ABB RobotStudio station: Welding_2.rspag

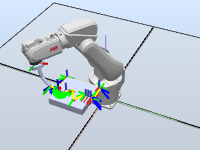
--- station ---
Station Welding_1 (saved by RobotStudio 20.1.9014.1)
Controller Controller2
  mechanical unit ROB_1: IRB120_3_58__01, 6 joints, base frame (0, 0, 0) mm
Layout (positions relative to the parent item):
  - IRB120_3_58__01 [mechanism, from Robots\IRB120_3_58_G_01.rslib] at (0, 0, 0) mm; joint values [-0.5429, 0.6455, -0.6027, 0.2244, 1.6631, 1.0335] (rad or m)
  - AssemblyWeldingTorch (2)_2 [part] at (431.78, -161.71, 537.76) mm, rotated rx -105 ry 0 rz -180 deg
  - Task1_Part1_2 [part] at (400, -100, 350) mm, rotated rx 90 ry 0 rz 0 deg
  - Task1_Part2 [part] at (300, -100, 350) mm, rotated rx 90 ry 0 rz 0 deg
  - Frame_1 [frame] at (400, 100, 370) mm
  - Frame_5 [frame] at (300, 100, 370) mm
  - Frame_6 [frame] at (300, -100, 370) mm
  - Frame_9 [frame] at (400, 85, 370) mm
  - Frame_10 [frame] at (400, 70, 370) mm
  - Frame_11 [frame] at (400, -50, 370) mm
Attachment: AssemblyWeldingTorch (2)_2 is attached to IRB120_3_58__01 / Link6

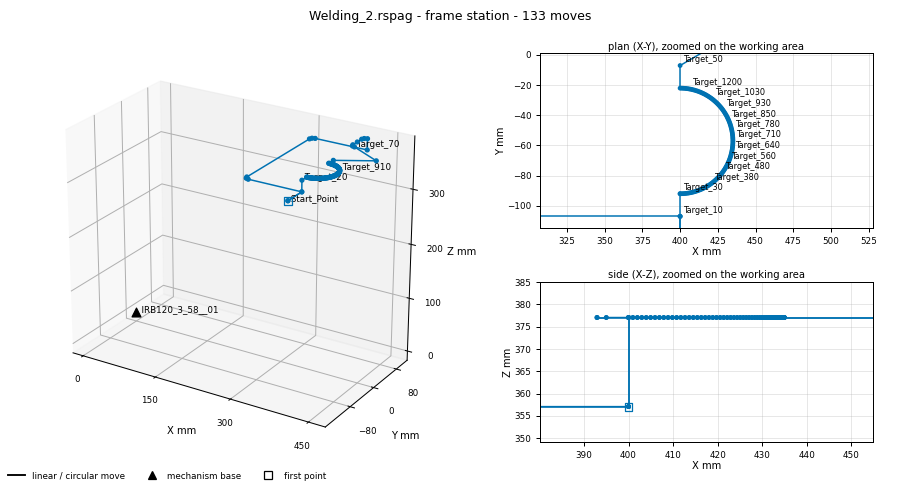
[picture p0: tool path of Welding_2.rspag in frame station, 133 of 133 moves have a stored position in this frame; points joined in program order, loops and branches not executed]
--- Backups/Controller2/RAPID/TASK1/PROGMOD/CalibData.mod ---
MODULE CalibData
    TASK PERS tooldata Tooldata_1:=[TRUE,[[35,0,150.231],[0.866025404,0,-0.5,0]],[1,[0,0,1],[1,0,0,0],0,0,0]];
    TASK PERS wobjdata weldPlate_1:=[FALSE,TRUE,"",[[400,-100,350],[1,0,0,0]],[[0,0,0],[1,0,0,0]]];
ENDMODULE

--- Backups/Controller2/RAPID/TASK1/PROGMOD/Module1.mod ---
MODULE Module1
        CONST robtarget Start_Point:=[[0,-50,7.071067812],[0.27059805,0.653281482,0.653281482,-0.27059805],[-1,0,0,0],[9E+09,9E+09,9E+09,9E+09,9E+09,9E+09]];
    CONST robtarget Target_10:=[[0,-7.071,7.071067812],[0.27059805,0.653281482,0.653281482,-0.27059805],[-1,0,0,0],[9E+09,9E+09,9E+09,9E+09,9E+09,9E+09]];
    CONST robtarget Target_20:=[[0,-7.071,27.071067812],[0.27059805,0.653281482,0.653281482,-0.27059805],[-1,0,0,0],[9E+09,9E+09,9E+09,9E+09,9E+09,9E+09]];
    CONST robtarget Target_30:=[[0,7.929,27.071067812],[0.27059805,0.653281482,0.653281482,-0.27059805],[-1,0,0,0],[9E+09,9E+09,9E+09,9E+09,9E+09,9E+09]];
    CONST robtarget Target_40:=[[0,77.929,27.071067812],[0.27059805,0.653281482,0.653281482,-0.27059805],[-1,0,0,0],[9E+09,9E+09,9E+09,9E+09,9E+09,9E+09]];
    CONST robtarget Target_50:=[[0,92.929,27.071067812],[0.27059805,0.653281482,0.653281482,-0.27059805],[-1,0,0,0],[9E+09,9E+09,9E+09,9E+09,9E+09,9E+09]];
    CONST robtarget Target_60:=[[60,127.929,27.071067812],[0.27059805,0.653281482,0.653281482,-0.27059805],[-1,0,0,0],[9E+09,9E+09,9E+09,9E+09,9E+09,9E+09]];
    CONST robtarget Target_70:=[[0,162.929,27.071067812],[0.27059805,0.653281482,0.653281482,-0.27059805],[-1,0,0,0],[9E+09,9E+09,9E+09,9E+09,9E+09,9E+09]];
    CONST robtarget Target_90:=[[0,207.071,7.071067812],[0.27059805,-0.653281482,0.653281482,0.27059805],[0,-1,3,0],[9E+09,9E+09,9E+09,9E+09,9E+09,9E+09]];
    CONST robtarget Target_100:=[[-100,207.071,7.071067812],[0.27059805,-0.653281482,0.653281482,0.27059805],[0,-1,3,0],[9E+09,9E+09,9E+09,9E+09,9E+09,9E+09]];
    CONST robtarget Target_110:=[[-107.071,200,7.071067812],[0,0.923879532,0,-0.382683432],[0,-1,2,0],[9E+09,9E+09,9E+09,9E+09,9E+09,9E+09]];
    CONST robtarget Target_120:=[[-107.071,0,7.071],[0,0.923879533,0,-0.382683432],[-1,0,1,0],[9E+09,9E+09,9E+09,9E+09,9E+09,9E+09]];
    CONST robtarget Target_130:=[[-100,-7.071,7.071],[0.27059805,0.653281483,0.653281483,-0.27059805],[-1,0,0,0],[9E+09,9E+09,9E+09,9E+09,9E+09,9E+09]];
    CONST robtarget Target_140:=[[0,-7.071,7.071067812],[0.27059805,0.653281482,0.653281482,-0.27059805],[-1,0,0,0],[9E+09,9E+09,9E+09,9E+09,9E+09,9E+09]];
    CONST robtarget Target_150:=[[-2,-9.698,8.29],[0.699810239,0.292325175,0.577022876,0.303077913],[-1,0,-1,0],[9E+09,9E+09,9E+09,9E+09,9E+09,9E+09]];
    CONST robtarget End_Point:=[[0,-50,0],[0.27059805,0.653281482,0.653281482,-0.27059805],[-1,0,0,0],[9E+09,9E+09,9E+09,9E+09,9E+09,9E+09]];
    CONST robtarget Target_30_1:=[[35,42.928932188,27.071067812],[0.27059805,0.653281482,0.653281482,-0.27059805],[-1,0,0,0],[9E+09,9E+09,9E+09,9E+09,9E+09,9E+09]];
    CONST robtarget Target_30_4:=[[32.122,36.212,30],[0.699810239,0.292325175,0.577022876,0.303077913],[-1,0,-1,0],[9E+09,9E+09,9E+09,9E+09,9E+09,9E+09]];
    CONST robtarget Target_30_5:=[[26.122,57.788,30],[0.699810239,0.292325175,0.577022876,0.303077913],[-1,0,-1,0],[9E+09,9E+09,9E+09,9E+09,9E+09,9E+09]];
    CONST robtarget Target_30_6:=[[7.364,71.822,30],[0.699810239,0.292325175,0.577022876,0.303077913],[-1,0,-1,0],[9E+09,9E+09,9E+09,9E+09,9E+09,9E+09]];
    CONST robtarget Target_30_7:=[[-2.5,81.534,30],[0.699810239,0.292325175,0.577022876,0.303077913],[-1,0,-1,0],[9E+09,9E+09,9E+09,9E+09,9E+09,9E+09]];
    CONST robtarget Target_30_8:=[[-2.5,88,30],[0.699810239,0.292325175,0.577022876,0.303077913],[-1,0,-1,0],[9E+09,9E+09,9E+09,9E+09,9E+09,9E+09]];
    CONST robtarget Target_30_3:=[[27.364,20.178,30],[0.699810239,0.292325175,0.577022876,0.303077913],[-1,0,-1,0],[9E+09,9E+09,9E+09,9E+09,9E+09,9E+09]];
    CONST robtarget Target_80:=[[-7.071067812,200,27.071],[0,0.923879532,0,-0.382683432],[0,-1,2,0],[9E+09,9E+09,9E+09,9E+09,9E+09,9E+09]];
    CONST robtarget Target_30_2:=[[15.186,8.466,30],[0.699810239,0.292325175,0.577022876,0.303077913],[-1,0,-1,0],[9E+09,9E+09,9E+09,9E+09,9E+09,9E+09]];
    CONST robtarget Target_70_2:=[[-5,165.000095901,27.071],[0.146446609,0.853553391,0.353553391,-0.35355339],[0,0,1,0],[9E+09,9E+09,9E+09,9E+09,9E+09,9E+09]];
    CONST robtarget Target_70_2_2:=[[-7.071,170.000067812,27.071],[0,0.923879533,0,-0.382683432],[0,-1,2,0],[9E+09,9E+09,9E+09,9E+09,9E+09,9E+09]];
    CONST robtarget Target_70_3:=[[-7.071067812,185,27.071],[0,0.923879533,0,-0.382683432],[0,-1,2,0],[9E+09,9E+09,9E+09,9E+09,9E+09,9E+09]];
    CONST robtarget Target_80_3:=[[-5,205,27.071],[0.146446609,-0.853553391,0.353553391,0.353553391],[0,-1,2,0],[9E+09,9E+09,9E+09,9E+09,9E+09,9E+09]];
    CONST robtarget Target_80_4:=[[0,207.071067812,27.071],[0.27059805,-0.653281482,0.653281482,0.27059805],[0,-1,3,0],[9E+09,9E+09,9E+09,9E+09,9E+09,9E+09]];
    CONST robtarget Target_100_3:=[[-104.99995205,204.99995205,7.071067812],[0.146446609,-0.853553391,0.353553391,0.353553391],[0,-1,2,0],[9E+09,9E+09,9E+09,9E+09,9E+09,9E+09]];
    CONST robtarget Target_120_3:=[[-104.99995205,-4.99995205,7.071],[0.146446609,0.853553391,0.353553391,-0.35355339],[-1,0,1,0],[9E+09,9E+09,9E+09,9E+09,9E+09,9E+09]];
    CONST robtarget zEnd_Point:=[[0,-50,7.071067812],[0.27059805,0.653281482,0.653281482,-0.27059805],[-1,0,0,0],[9E+09,9E+09,9E+09,9E+09,9E+09,9E+09]];
    CONST robtarget Target_170:=[[0.999863951,7.94321693,27.071067812],[0.27059805,0.653281482,0.653281482,-0.27059805],[-1,0,0,0],[9E+09,9E+09,9E+09,9E+09,9E+09,9E+09]];
    CONST robtarget Target_180:=[[1.998911742,7.986059498,27.071067812],[0.27059805,0.653281482,0.653281482,-0.27059805],[-1,0,0,0],[9E+09,9E+09,9E+09,9E+09,9E+09,9E+09]];
    CONST robtarget Target_190:=[[2.99632788,8.057424919,27.071067812],[0.27059805,0.653281482,0.653281482,-0.27059805],[-1,0,0,0],[9E+09,9E+09,9E+09,9E+09,9E+09,9E+09]];
    CONST robtarget Target_200:=[[3.991298202,8.15725494,27.071067812],[0.27059805,0.653281482,0.653281482,-0.27059805],[-1,0,0,0],[9E+09,9E+09,9E+09,9E+09,9E+09,9E+09]];
    CONST robtarget Target_210:=[[4.983010543,8.285468072,27.071067812],[0.27059805,0.653281482,0.653281482,-0.27059805],[-1,0,0,0],[9E+09,9E+09,9E+09,9E+09,9E+09,9E+09]];
    CONST robtarget Target_220:=[[5.970655397,8.44195966,27.071067812],[0.27059805,0.653281482,0.653281482,-0.27059805],[-1,0,0,0],[9E+09,9E+09,9E+09,9E+09,9E+09,9E+09]];
    CONST robtarget Target_230:=[[6.953426578,8.626601964,27.071067812],[0.27059805,0.653281482,0.653281482,-0.27059805],[-1,0,0,0],[9E+09,9E+09,9E+09,9E+09,9E+09,9E+09]];
    CONST robtarget Target_240:=[[7.930521878,8.839244264,27.071067812],[0.27059805,0.653281482,0.653281482,-0.27059805],[-1,0,0,0],[9E+09,9E+09,9E+09,9E+09,9E+09,9E+09]];
    CONST robtarget Target_250:=[[8.901143724,9.079712989,27.071067812],[0.27059805,0.653281482,0.653281482,-0.27059805],[-1,0,0,0],[9E+09,9E+09,9E+09,9E+09,9E+09,9E+09]];
    CONST robtarget Target_260:=[[9.864499824,9.347811849,27.071067812],[0.27059805,0.653281482,0.653281482,-0.27059805],[-1,0,0,0],[9E+09,9E+09,9E+09,9E+09,9E+09,9E+09]];
    CONST robtarget Target_270:=[[10.819803819,9.643322004,27.071067812],[0.27059805,0.653281482,0.653281482,-0.27059805],[-1,0,0,0],[9E+09,9E+09,9E+09,9E+09,9E+09,9E+09]];
    CONST robtarget Target_280:=[[11.766275922,9.966002237,27.071067812],[0.27059805,0.653281482,0.653281482,-0.27059805],[-1,0,0,0],[9E+09,9E+09,9E+09,9E+09,9E+09,9E+09]];
    CONST robtarget Target_290:=[[12.703143555,10.315589155,27.071067812],[0.27059805,0.653281482,0.653281482,-0.27059805],[-1,0,0,0],[9E+09,9E+09,9E+09,9E+09,9E+09,9E+09]];
    CONST robtarget Target_300:=[[13.629641981,10.691797398,27.071067812],[0.27059805,0.653281482,0.653281482,-0.27059805],[-1,0,0,0],[9E+09,9E+09,9E+09,9E+09,9E+09,9E+09]];
    CONST robtarget Target_310:=[[14.545014925,11.094319879,27.071067812],[0.27059805,0.653281482,0.653281482,-0.27059805],[-1,0,0,0],[9E+09,9E+09,9E+09,9E+09,9E+09,9E+09]];
    CONST robtarget Target_320:=[[15.448515195,11.522828032,27.071067812],[0.27059805,0.653281482,0.653281482,-0.27059805],[-1,0,0,0],[9E+09,9E+09,9E+09,9E+09,9E+09,9E+09]];
    CONST robtarget Target_330:=[[16.33940529,11.976972076,27.071067812],[0.27059805,0.653281482,0.653281482,-0.27059805],[-1,0,0,0],[9E+09,9E+09,9E+09,9E+09,9E+09,9E+09]];
    CONST robtarget Target_340:=[[17.216958002,12.456381308,27.071067812],[0.27059805,0.653281482,0.653281482,-0.27059805],[-1,0,0,0],[9E+09,9E+09,9E+09,9E+09,9E+09,9E+09]];
    CONST robtarget Target_350:=[[18.080457011,12.960664399,27.071067812],[0.27059805,0.653281482,0.653281482,-0.27059805],[-1,0,0,0],[9E+09,9E+09,9E+09,9E+09,9E+09,9E+09]];
    CONST robtarget Target_360:=[[18.929197468,13.489409718,27.071067812],[0.27059805,0.653281482,0.653281482,-0.27059805],[-1,0,0,0],[9E+09,9E+09,9E+09,9E+09,9E+09,9E+09]];
    CONST robtarget Target_370:=[[19.762486569,14.042185666,27.071067812],[0.27059805,0.653281482,0.653281482,-0.27059805],[-1,0,0,0],[9E+09,9E+09,9E+09,9E+09,9E+09,9E+09]];
    CONST robtarget Target_380:=[[20.579644125,14.618541027,27.071067812],[0.27059805,0.653281482,0.653281482,-0.27059805],[-1,0,0,0],[9E+09,9E+09,9E+09,9E+09,9E+09,9E+09]];
    CONST robtarget Target_390:=[[21.380003115,15.21800534,27.071067812],[0.27059805,0.653281482,0.653281482,-0.27059805],[-1,0,0,0],[9E+09,9E+09,9E+09,9E+09,9E+09,9E+09]];
    CONST robtarget Target_400:=[[22.162910229,15.840089278,27.071067812],[0.27059805,0.653281482,0.653281482,-0.27059805],[-1,0,0,0],[9E+09,9E+09,9E+09,9E+09,9E+09,9E+09]];
    CONST robtarget Target_410:=[[22.927726401,16.484285053,27.071067812],[0.27059805,0.653281482,0.653281482,-0.27059805],[-1,0,0,0],[9E+09,9E+09,9E+09,9E+09,9E+09,9E+09]];
    CONST robtarget Target_420:=[[23.673827336,17.150066827,27.071067812],[0.27059805,0.653281482,0.653281482,-0.27059805],[-1,0,0,0],[9E+09,9E+09,9E+09,9E+09,9E+09,9E+09]];
    CONST robtarget Target_430:=[[24.400604011,17.836891141,27.071067812],[0.27059805,0.653281482,0.653281482,-0.27059805],[-1,0,0,0],[9E+09,9E+09,9E+09,9E+09,9E+09,9E+09]];
    CONST robtarget Target_440:=[[25.107463181,18.544197361,27.071067812],[0.27059805,0.653281482,0.653281482,-0.27059805],[-1,0,0,0],[9E+09,9E+09,9E+09,9E+09,9E+09,9E+09]];
    CONST robtarget Target_450:=[[25.793827858,19.271408132,27.071067812],[0.27059805,0.653281482,0.653281482,-0.27059805],[-1,0,0,0],[9E+09,9E+09,9E+09,9E+09,9E+09,9E+09]];
    CONST robtarget Target_460:=[[26.45913778,20.017929854,27.071067812],[0.27059805,0.653281482,0.653281482,-0.27059805],[-1,0,0,0],[9E+09,9E+09,9E+09,9E+09,9E+09,9E+09]];
    CONST robtarget Target_470:=[[27.102849876,20.783153163,27.071067812],[0.27059805,0.653281482,0.653281482,-0.27059805],[-1,0,0,0],[9E+09,9E+09,9E+09,9E+09,9E+09,9E+09]];
    CONST robtarget Target_480:=[[27.724438701,21.566453429,27.071067812],[0.27059805,0.653281482,0.653281482,-0.27059805],[-1,0,0,0],[9E+09,9E+09,9E+09,9E+09,9E+09,9E+09]];
    CONST robtarget Target_490:=[[28.323396871,22.367191267,27.071067812],[0.27059805,0.653281482,0.653281482,-0.27059805],[-1,0,0,0],[9E+09,9E+09,9E+09,9E+09,9E+09,9E+09]];
    CONST robtarget Target_500:=[[28.899235474,23.184713058,27.071067812],[0.27059805,0.653281482,0.653281482,-0.27059805],[-1,0,0,0],[9E+09,9E+09,9E+09,9E+09,9E+09,9E+09]];
    CONST robtarget Target_510:=[[29.451484468,24.018351483,27.071067812],[0.27059805,0.653281482,0.653281482,-0.27059805],[-1,0,0,0],[9E+09,9E+09,9E+09,9E+09,9E+09,9E+09]];
    CONST robtarget Target_520:=[[29.97969307,24.867426066,27.071067812],[0.27059805,0.653281482,0.653281482,-0.27059805],[-1,0,0,0],[9E+09,9E+09,9E+09,9E+09,9E+09,9E+09]];
    CONST robtarget Target_530:=[[30.483430118,25.731243732,27.071067812],[0.27059805,0.653281482,0.653281482,-0.27059805],[-1,0,0,0],[9E+09,9E+09,9E+09,9E+09,9E+09,9E+09]];
    CONST robtarget Target_540:=[[30.962284426,26.609099373,27.071067812],[0.27059805,0.653281482,0.653281482,-0.27059805],[-1,0,0,0],[9E+09,9E+09,9E+09,9E+09,9E+09,9E+09]];
    CONST robtarget Target_550:=[[31.415865119,27.50027642,27.071067812],[0.27059805,0.653281482,0.653281482,-0.27059805],[-1,0,0,0],[9E+09,9E+09,9E+09,9E+09,9E+09,9E+09]];
    CONST robtarget Target_560:=[[31.843801953,28.404047432,27.071067812],[0.27059805,0.653281482,0.653281482,-0.27059805],[-1,0,0,0],[9E+09,9E+09,9E+09,9E+09,9E+09,9E+09]];
    CONST robtarget Target_570:=[[32.245745614,29.319674685,27.071067812],[0.27059805,0.653281482,0.653281482,-0.27059805],[-1,0,0,0],[9E+09,9E+09,9E+09,9E+09,9E+09,9E+09]];
    CONST robtarget Target_580:=[[32.621368009,30.246410781,27.071067812],[0.27059805,0.653281482,0.653281482,-0.27059805],[-1,0,0,0],[9E+09,9E+09,9E+09,9E+09,9E+09,9E+09]];
    CONST robtarget Target_590:=[[32.970362527,31.183499252,27.071067812],[0.27059805,0.653281482,0.653281482,-0.27059805],[-1,0,0,0],[9E+09,9E+09,9E+09,9E+09,9E+09,9E+09]];
    CONST robtarget Target_600:=[[33.292444294,32.130175178,27.071067812],[0.27059805,0.653281482,0.653281482,-0.27059805],[-1,0,0,0],[9E+09,9E+09,9E+09,9E+09,9E+09,9E+09]];
    CONST robtarget Target_610:=[[33.587350404,33.085665817,27.071067812],[0.27059805,0.653281482,0.653281482,-0.27059805],[-1,0,0,0],[9E+09,9E+09,9E+09,9E+09,9E+09,9E+09]];
    CONST robtarget Target_620:=[[33.854840134,34.049191229,27.071067812],[0.27059805,0.653281482,0.653281482,-0.27059805],[-1,0,0,0],[9E+09,9E+09,9E+09,9E+09,9E+09,9E+09]];
    CONST robtarget Target_630:=[[34.09469514,35.019964915,27.071067812],[0.27059805,0.653281482,0.653281482,-0.27059805],[-1,0,0,0],[9E+09,9E+09,9E+09,9E+09,9E+09,9E+09]];
    CONST robtarget Target_640:=[[34.306719635,35.997194463,27.071067812],[0.27059805,0.653281482,0.653281482,-0.27059805],[-1,0,0,0],[9E+09,9E+09,9E+09,9E+09,9E+09,9E+09]];
    CONST robtarget Target_650:=[[34.49074055,36.980082186,27.071067812],[0.27059805,0.653281482,0.653281482,-0.27059805],[-1,0,0,0],[9E+09,9E+09,9E+09,9E+09,9E+09,9E+09]];
    CONST robtarget Target_660:=[[34.646607673,37.967825784,27.071067812],[0.27059805,0.653281482,0.653281482,-0.27059805],[-1,0,0,0],[9E+09,9E+09,9E+09,9E+09,9E+09,9E+09]];
    CONST robtarget Target_670:=[[34.774193775,38.959618989,27.071067812],[0.27059805,0.653281482,0.653281482,-0.27059805],[-1,0,0,0],[9E+09,9E+09,9E+09,9E+09,9E+09,9E+09]];
    CONST robtarget Target_680:=[[34.873394712,39.954652229,27.071067812],[0.27059805,0.653281482,0.653281482,-0.27059805],[-1,0,0,0],[9E+09,9E+09,9E+09,9E+09,9E+09,9E+09]];
    CONST robtarget Target_690:=[[34.944129507,40.952113287,27.071067812],[0.27059805,0.653281482,0.653281482,-0.27059805],[-1,0,0,0],[9E+09,9E+09,9E+09,9E+09,9E+09,9E+09]];
    CONST robtarget Target_700:=[[34.986340424,41.951187966,27.071067812],[0.27059805,0.653281482,0.653281482,-0.27059805],[-1,0,0,0],[9E+09,9E+09,9E+09,9E+09,9E+09,9E+09]];
    CONST robtarget Target_710:=[[34.999993005,42.951060749,27.071067812],[0.27059805,0.653281482,0.653281482,-0.27059805],[-1,0,0,0],[9E+09,9E+09,9E+09,9E+09,9E+09,9E+09]];
    CONST robtarget Target_720:=[[34.985076106,43.950915469,27.071067812],[0.27059805,0.653281482,0.653281482,-0.27059805],[-1,0,0,0],[9E+09,9E+09,9E+09,9E+09,9E+09,9E+09]];
    CONST robtarget Target_730:=[[34.941601905,44.949935973,27.071067812],[0.27059805,0.653281482,0.653281482,-0.27059805],[-1,0,0,0],[9E+09,9E+09,9E+09,9E+09,9E+09,9E+09]];
    CONST robtarget Target_740:=[[34.869605888,45.947306791,27.071067812],[0.27059805,0.653281482,0.653281482,-0.27059805],[-1,0,0,0],[9E+09,9E+09,9E+09,9E+09,9E+09,9E+09]];
    CONST robtarget Target_750:=[[34.769146822,46.942213797,27.071067812],[0.27059805,0.653281482,0.653281482,-0.27059805],[-1,0,0,0],[9E+09,9E+09,9E+09,9E+09,9E+09,9E+09]];
    CONST robtarget Target_760:=[[34.64030671,47.933844878,27.071067812],[0.27059805,0.653281482,0.653281482,-0.27059805],[-1,0,0,0],[9E+09,9E+09,9E+09,9E+09,9E+09,9E+09]];
    CONST robtarget Target_770:=[[34.48319072,48.921390593,27.071067812],[0.27059805,0.653281482,0.653281482,-0.27059805],[-1,0,0,0],[9E+09,9E+09,9E+09,9E+09,9E+09,9E+09]];
    CONST robtarget Target_780:=[[34.297927102,49.904044839,27.071067812],[0.27059805,0.653281482,0.653281482,-0.27059805],[-1,0,0,0],[9E+09,9E+09,9E+09,9E+09,9E+09,9E+09]];
    CONST robtarget Target_790:=[[34.084667081,50.881005502,27.071067812],[0.27059805,0.653281482,0.653281482,-0.27059805],[-1,0,0,0],[9E+09,9E+09,9E+09,9E+09,9E+09,9E+09]];
    CONST robtarget Target_800:=[[33.843584734,51.851475119,27.071067812],[0.27059805,0.653281482,0.653281482,-0.27059805],[-1,0,0,0],[9E+09,9E+09,9E+09,9E+09,9E+09,9E+09]];
    CONST robtarget Target_810:=[[33.574876851,52.814661522,27.071067812],[0.27059805,0.653281482,0.653281482,-0.27059805],[-1,0,0,0],[9E+09,9E+09,9E+09,9E+09,9E+09,9E+09]];
    CONST robtarget Target_820:=[[33.278762769,53.769778492,27.071067812],[0.27059805,0.653281482,0.653281482,-0.27059805],[-1,0,0,0],[9E+09,9E+09,9E+09,9E+09,9E+09,9E+09]];
    CONST robtarget Target_830:=[[32.955484198,54.716046393,27.071067812],[0.27059805,0.653281482,0.653281482,-0.27059805],[-1,0,0,0],[9E+09,9E+09,9E+09,9E+09,9E+09,9E+09]];
    CONST robtarget Target_840:=[[32.605305021,55.652692814,27.071067812],[0.27059805,0.653281482,0.653281482,-0.27059805],[-1,0,0,0],[9E+09,9E+09,9E+09,9E+09,9E+09,9E+09]];
    CONST robtarget Target_850:=[[32.22851108,56.578953199,27.071067812],[0.27059805,0.653281482,0.653281482,-0.27059805],[-1,0,0,0],[9E+09,9E+09,9E+09,9E+09,9E+09,9E+09]];
    CONST robtarget Target_860:=[[31.825409939,57.494071467,27.071067812],[0.27059805,0.653281482,0.653281482,-0.27059805],[-1,0,0,0],[9E+09,9E+09,9E+09,9E+09,9E+09,9E+09]];
    CONST robtarget Target_870:=[[31.396330639,58.397300635,27.071067812],[0.27059805,0.653281482,0.653281482,-0.27059805],[-1,0,0,0],[9E+09,9E+09,9E+09,9E+09,9E+09,9E+09]];
    CONST robtarget Target_880:=[[30.941623425,59.287903422,27.071067812],[0.27059805,0.653281482,0.653281482,-0.27059805],[-1,0,0,0],[9E+09,9E+09,9E+09,9E+09,9E+09,9E+09]];
    CONST robtarget Target_890:=[[30.461659461,60.165152855,27.071067812],[0.27059805,0.653281482,0.653281482,-0.27059805],[-1,0,0,0],[9E+09,9E+09,9E+09,9E+09,9E+09,9E+09]];
    CONST robtarget Target_900:=[[29.956830528,61.028332861,27.071067812],[0.27059805,0.653281482,0.653281482,-0.27059805],[-1,0,0,0],[9E+09,9E+09,9E+09,9E+09,9E+09,9E+09]];
    CONST robtarget Target_910:=[[29.427548703,61.876738851,27.071067812],[0.27059805,0.653281482,0.653281482,-0.27059805],[-1,0,0,0],[9E+09,9E+09,9E+09,9E+09,9E+09,9E+09]];
    CONST robtarget Target_920:=[[28.874246023,62.709678296,27.071067812],[0.27059805,0.653281482,0.653281482,-0.27059805],[-1,0,0,0],[9E+09,9E+09,9E+09,9E+09,9E+09,9E+09]];
    CONST robtarget Target_930:=[[28.297374134,63.526471292,27.071067812],[0.27059805,0.653281482,0.653281482,-0.27059805],[-1,0,0,0],[9E+09,9E+09,9E+09,9E+09,9E+09,9E+09]];
    CONST robtarget Target_940:=[[27.697403918,64.326451114,27.071067812],[0.27059805,0.653281482,0.653281482,-0.27059805],[-1,0,0,0],[9E+09,9E+09,9E+09,9E+09,9E+09,9E+09]];
    CONST robtarget Target_950:=[[27.074825116,65.108964762,27.071067812],[0.27059805,0.653281482,0.653281482,-0.27059805],[-1,0,0,0],[9E+09,9E+09,9E+09,9E+09,9E+09,9E+09]];
    CONST robtarget Target_960:=[[26.430145918,65.873373492,27.071067812],[0.27059805,0.653281482,0.653281482,-0.27059805],[-1,0,0,0],[9E+09,9E+09,9E+09,9E+09,9E+09,9E+09]];
    CONST robtarget Target_970:=[[25.763892559,66.61905334,27.071067812],[0.27059805,0.653281482,0.653281482,-0.27059805],[-1,0,0,0],[9E+09,9E+09,9E+09,9E+09,9E+09,9E+09]];
    CONST robtarget Target_980:=[[25.076608882,67.34539563,27.071067812],[0.27059805,0.653281482,0.653281482,-0.27059805],[-1,0,0,0],[9E+09,9E+09,9E+09,9E+09,9E+09,9E+09]];
    CONST robtarget Target_990:=[[24.368855896,68.051807468,27.071067812],[0.27059805,0.653281482,0.653281482,-0.27059805],[-1,0,0,0],[9E+09,9E+09,9E+09,9E+09,9E+09,9E+09]];
    CONST robtarget Target_1000:=[[23.641211319,68.737712232,27.071067812],[0.27059805,0.653281482,0.653281482,-0.27059805],[-1,0,0,0],[9E+09,9E+09,9E+09,9E+09,9E+09,9E+09]];
    CONST robtarget Target_1010:=[[22.894269108,69.402550037,27.071067812],[0.27059805,0.653281482,0.653281482,-0.27059805],[-1,0,0,0],[9E+09,9E+09,9E+09,9E+09,9E+09,9E+09]];
    CONST robtarget Target_1020:=[[22.128638968,70.045778196,27.071067812],[0.27059805,0.653281482,0.653281482,-0.27059805],[-1,0,0,0],[9E+09,9E+09,9E+09,9E+09,9E+09,9E+09]];
    CONST robtarget Target_1030:=[[21.344945862,70.66687166,27.071067812],[0.27059805,0.653281482,0.653281482,-0.27059805],[-1,0,0,0],[9E+09,9E+09,9E+09,9E+09,9E+09,9E+09]];
    CONST robtarget Target_1040:=[[20.543829496,71.265323448,27.071067812],[0.27059805,0.653281482,0.653281482,-0.27059805],[-1,0,0,0],[9E+09,9E+09,9E+09,9E+09,9E+09,9E+09]];
    CONST robtarget Target_1050:=[[19.725943798,71.840645061,27.071067812],[0.27059805,0.653281482,0.653281482,-0.27059805],[-1,0,0,0],[9E+09,9E+09,9E+09,9E+09,9E+09,9E+09]];
    CONST robtarget Target_1060:=[[18.891956384,72.392366882,27.071067812],[0.27059805,0.653281482,0.653281482,-0.27059805],[-1,0,0,0],[9E+09,9E+09,9E+09,9E+09,9E+09,9E+09]];
    CONST robtarget Target_1070:=[[18.042548014,72.920038556,27.071067812],[0.27059805,0.653281482,0.653281482,-0.27059805],[-1,0,0,0],[9E+09,9E+09,9E+09,9E+09,9E+09,9E+09]];
    CONST robtarget Target_1080:=[[17.178412035,73.423229359,27.071067812],[0.27059805,0.653281482,0.653281482,-0.27059805],[-1,0,0,0],[9E+09,9E+09,9E+09,9E+09,9E+09,9E+09]];
    CONST robtarget Target_1090:=[[16.300253816,73.901528552,27.071067812],[0.27059805,0.653281482,0.653281482,-0.27059805],[-1,0,0,0],[9E+09,9E+09,9E+09,9E+09,9E+09,9E+09]];
    CONST robtarget Target_1100:=[[15.408790173,74.354545713,27.071067812],[0.27059805,0.653281482,0.653281482,-0.27059805],[-1,0,0,0],[9E+09,9E+09,9E+09,9E+09,9E+09,9E+09]];
    CONST robtarget Target_1110:=[[14.504748782,74.781911056,27.071067812],[0.27059805,0.653281482,0.653281482,-0.27059805],[-1,0,0,0],[9E+09,9E+09,9E+09,9E+09,9E+09,9E+09]];
    CONST robtarget Target_1120:=[[13.588867584,75.183275737,27.071067812],[0.27059805,0.653281482,0.653281482,-0.27059805],[-1,0,0,0],[9E+09,9E+09,9E+09,9E+09,9E+09,9E+09]];
    CONST robtarget Target_1130:=[[12.661894188,75.558312132,27.071067812],[0.27059805,0.653281482,0.653281482,-0.27059805],[-1,0,0,0],[9E+09,9E+09,9E+09,9E+09,9E+09,9E+09]];
    CONST robtarget Target_1140:=[[11.724585255,75.906714111,27.071067812],[0.27059805,0.653281482,0.653281482,-0.27059805],[-1,0,0,0],[9E+09,9E+09,9E+09,9E+09,9E+09,9E+09]];
    CONST robtarget Target_1150:=[[10.777705884,76.228197283,27.071067812],[0.27059805,0.653281482,0.653281482,-0.27059805],[-1,0,0,0],[9E+09,9E+09,9E+09,9E+09,9E+09,9E+09]];
    CONST robtarget Target_1160:=[[9.822028983,76.522499231,27.071067812],[0.27059805,0.653281482,0.653281482,-0.27059805],[-1,0,0,0],[9E+09,9E+09,9E+09,9E+09,9E+09,9E+09]];
    CONST robtarget Target_1170:=[[8.858334645,76.789379724,27.071067812],[0.27059805,0.653281482,0.653281482,-0.27059805],[-1,0,0,0],[9E+09,9E+09,9E+09,9E+09,9E+09,9E+09]];
    CONST robtarget Target_1180:=[[7.887409505,77.028620915,27.071067812],[0.27059805,0.653281482,0.653281482,-0.27059805],[-1,0,0,0],[9E+09,9E+09,9E+09,9E+09,9E+09,9E+09]];
    CONST robtarget Target_1190:=[[6.910046102,77.24002752,27.071067812],[0.27059805,0.653281482,0.653281482,-0.27059805],[-1,0,0,0],[9E+09,9E+09,9E+09,9E+09,9E+09,9E+09]];
    CONST robtarget Target_1200:=[[5.927042228,77.423426972,27.071067812],[0.27059805,0.653281482,0.653281482,-0.27059805],[-1,0,0,0],[9E+09,9E+09,9E+09,9E+09,9E+09,9E+09]];
    CONST robtarget Target_1210:=[[4.939200282,77.578669569,27.071067812],[0.27059805,0.653281482,0.653281482,-0.27059805],[-1,0,0,0],[9E+09,9E+09,9E+09,9E+09,9E+09,9E+09]];
    CONST robtarget Target_1220:=[[3.94732661,77.70562859,27.071067812],[0.27059805,0.653281482,0.653281482,-0.27059805],[-1,0,0,0],[9E+09,9E+09,9E+09,9E+09,9E+09,9E+09]];
    CONST robtarget Target_1230:=[[2.952230849,77.804200402,27.071067812],[0.27059805,0.653281482,0.653281482,-0.27059805],[-1,0,0,0],[9E+09,9E+09,9E+09,9E+09,9E+09,9E+09]];
    CONST robtarget Target_1240:=[[1.954725269,77.874304544,27.071067812],[0.27059805,0.653281482,0.653281482,-0.27059805],[-1,0,0,0],[9E+09,9E+09,9E+09,9E+09,9E+09,9E+09]];
    CONST robtarget Target_1250:=[[0.955624102,77.915883792,27.071067812],[0.27059805,0.653281482,0.653281482,-0.27059805],[-1,0,0,0],[9E+09,9E+09,9E+09,9E+09,9E+09,9E+09]];
    CONST robtarget Target_160:=[[0,7.928932188,27.071067812],[0.27059805,0.653281482,0.653281482,-0.27059805],[-1,0,0,0],[9E+09,9E+09,9E+09,9E+09,9E+09,9E+09]];
!***********************************************************
    !
    ! Module:  Module1
    !
    ! Description:
    !   <Insert description here>
    !
    ! Author: Koldas2
    !
    ! Version: 1.0
    !
    !***********************************************************


    !***********************************************************
    !
    ! Procedure main
    !
    !   This is the entry point of your program
    !
    !***********************************************************
    PROC main()
        !Add your code here
        Path_10;
    ENDPROC
    PROC Path_10()
        MoveL Start_Point,v100,z1,Tooldata_1\WObj:=weldPlate_1;
        MoveL Target_10,v20,z1,Tooldata_1\WObj:=weldPlate_1;
        MoveL Target_20,v20,z1,Tooldata_1\WObj:=weldPlate_1;
        MoveL Target_30,v20,z1,Tooldata_1\WObj:=weldPlate_1;
        MoveL Target_160,v20,z1,Tooldata_1\WObj:=weldPlate_1;
        MoveL Target_170,v20,z1,Tooldata_1\WObj:=weldPlate_1;
        MoveL Target_180,v20,z1,Tooldata_1\WObj:=weldPlate_1;
        MoveL Target_190,v20,z1,Tooldata_1\WObj:=weldPlate_1;
        MoveL Target_200,v20,z1,Tooldata_1\WObj:=weldPlate_1;
        MoveL Target_210,v20,z1,Tooldata_1\WObj:=weldPlate_1;
        MoveL Target_220,v20,z1,Tooldata_1\WObj:=weldPlate_1;
        MoveL Target_230,v20,z1,Tooldata_1\WObj:=weldPlate_1;
        MoveL Target_240,v20,z1,Tooldata_1\WObj:=weldPlate_1;
        MoveL Target_250,v20,z1,Tooldata_1\WObj:=weldPlate_1;
        MoveL Target_260,v20,z1,Tooldata_1\WObj:=weldPlate_1;
        MoveL Target_270,v20,z1,Tooldata_1\WObj:=weldPlate_1;
        MoveL Target_280,v20,z1,Tooldata_1\WObj:=weldPlate_1;
        MoveL Target_290,v20,z1,Tooldata_1\WObj:=weldPlate_1;
        MoveL Target_300,v20,z1,Tooldata_1\WObj:=weldPlate_1;
        MoveL Target_310,v20,z1,Tooldata_1\WObj:=weldPlate_1;
        MoveL Target_320,v20,z1,Tooldata_1\WObj:=weldPlate_1;
        MoveL Target_330,v20,z1,Tooldata_1\WObj:=weldPlate_1;
        MoveL Target_340,v20,z1,Tooldata_1\WObj:=weldPlate_1;
        MoveL Target_350,v20,z1,Tooldata_1\WObj:=weldPlate_1;
        MoveL Target_360,v20,z1,Tooldata_1\WObj:=weldPlate_1;
        MoveL Target_370,v20,z1,Tooldata_1\WObj:=weldPlate_1;
        MoveL Target_380,v20,z1,Tooldata_1\WObj:=weldPlate_1;
        MoveL Target_390,v20,z1,Tooldata_1\WObj:=weldPlate_1;
        MoveL Target_400,v20,z1,Tooldata_1\WObj:=weldPlate_1;
        MoveL Target_410,v20,z1,Tooldata_1\WObj:=weldPlate_1;
        MoveL Target_420,v20,z1,Tooldata_1\WObj:=weldPlate_1;
        MoveL Target_430,v20,z1,Tooldata_1\WObj:=weldPlate_1;
        MoveL Target_440,v20,z1,Tooldata_1\WObj:=weldPlate_1;
        MoveL Target_450,v20,z1,Tooldata_1\WObj:=weldPlate_1;
        MoveL Target_460,v20,z1,Tooldata_1\WObj:=weldPlate_1;
        MoveL Target_470,v20,z1,Tooldata_1\WObj:=weldPlate_1;
        MoveL Target_480,v20,z1,Tooldata_1\WObj:=weldPlate_1;
        MoveL Target_490,v20,z1,Tooldata_1\WObj:=weldPlate_1;
        MoveL Target_500,v20,z1,Tooldata_1\WObj:=weldPlate_1;
        MoveL Target_510,v20,z1,Tooldata_1\WObj:=weldPlate_1;
        MoveL Target_520,v20,z1,Tooldata_1\WObj:=weldPlate_1;
        MoveL Target_530,v20,z1,Tooldata_1\WObj:=weldPlate_1;
        MoveL Target_540,v20,z1,Tooldata_1\WObj:=weldPlate_1;
        MoveL Target_550,v20,z1,Tooldata_1\WObj:=weldPlate_1;
        MoveL Target_560,v20,z1,Tooldata_1\WObj:=weldPlate_1;
        MoveL Target_570,v20,z1,Tooldata_1\WObj:=weldPlate_1;
        MoveL Target_580,v20,z1,Tooldata_1\WObj:=weldPlate_1;
        MoveL Target_590,v20,z1,Tooldata_1\WObj:=weldPlate_1;
        MoveL Target_600,v20,z1,Tooldata_1\WObj:=weldPlate_1;
        MoveL Target_610,v20,z1,Tooldata_1\WObj:=weldPlate_1;
        MoveL Target_620,v20,z1,Tooldata_1\WObj:=weldPlate_1;
        MoveL Target_630,v20,z1,Tooldata_1\WObj:=weldPlate_1;
        MoveL Target_640,v20,z1,Tooldata_1\WObj:=weldPlate_1;
        MoveL Target_650,v20,z1,Tooldata_1\WObj:=weldPlate_1;
        MoveL Target_660,v20,z1,Tooldata_1\WObj:=weldPlate_1;
        MoveL Target_670,v20,z1,Tooldata_1\WObj:=weldPlate_1;
        MoveL Target_680,v20,z1,Tooldata_1\WObj:=weldPlate_1;
        MoveL Target_690,v20,z1,Tooldata_1\WObj:=weldPlate_1;
        MoveL Target_700,v20,z1,Tooldata_1\WObj:=weldPlate_1;
        MoveL Target_710,v20,z1,Tooldata_1\WObj:=weldPlate_1;
        MoveL Target_720,v20,z1,Tooldata_1\WObj:=weldPlate_1;
        MoveL Target_730,v20,z1,Tooldata_1\WObj:=weldPlate_1;
        MoveL Target_740,v20,z1,Tooldata_1\WObj:=weldPlate_1;
        MoveL Target_750,v20,z1,Tooldata_1\WObj:=weldPlate_1;
        MoveL Target_760,v20,z1,Tooldata_1\WObj:=weldPlate_1;
        MoveL Target_770,v20,z1,Tooldata_1\WObj:=weldPlate_1;
        MoveL Target_780,v20,z1,Tooldata_1\WObj:=weldPlate_1;
        MoveL Target_790,v20,z1,Tooldata_1\WObj:=weldPlate_1;
        MoveL Target_800,v20,z1,Tooldata_1\WObj:=weldPlate_1;
        MoveL Target_810,v20,z1,Tooldata_1\WObj:=weldPlate_1;
        MoveL Target_820,v20,z1,Tooldata_1\WObj:=weldPlate_1;
        MoveL Target_830,v20,z1,Tooldata_1\WObj:=weldPlate_1;
        MoveL Target_840,v20,z1,Tooldata_1\WObj:=weldPlate_1;
        MoveL Target_850,v20,z1,Tooldata_1\WObj:=weldPlate_1;
        MoveL Target_860,v20,z1,Tooldata_1\WObj:=weldPlate_1;
        MoveL Target_870,v20,z1,Tooldata_1\WObj:=weldPlate_1;
        MoveL Target_880,v20,z1,Tooldata_1\WObj:=weldPlate_1;
        MoveL Target_890,v20,z1,Tooldata_1\WObj:=weldPlate_1;
        MoveL Target_900,v20,z1,Tooldata_1\WObj:=weldPlate_1;
        MoveL Target_910,v20,z1,Tooldata_1\WObj:=weldPlate_1;
        MoveL Target_920,v20,z1,Tooldata_1\WObj:=weldPlate_1;
        MoveL Target_930,v20,z1,Tooldata_1\WObj:=weldPlate_1;
        MoveL Target_940,v20,z1,Tooldata_1\WObj:=weldPlate_1;
        MoveL Target_950,v20,z1,Tooldata_1\WObj:=weldPlate_1;
        MoveL Target_960,v20,z1,Tooldata_1\WObj:=weldPlate_1;
        MoveL Target_970,v20,z1,Tooldata_1\WObj:=weldPlate_1;
        MoveL Target_980,v20,z1,Tooldata_1\WObj:=weldPlate_1;
        MoveL Target_990,v20,z1,Tooldata_1\WObj:=weldPlate_1;
        MoveL Target_1000,v20,z1,Tooldata_1\WObj:=weldPlate_1;
        MoveL Target_1010,v20,z1,Tooldata_1\WObj:=weldPlate_1;
        MoveL Target_1020,v20,z1,Tooldata_1\WObj:=weldPlate_1;
        MoveL Target_1030,v20,z1,Tooldata_1\WObj:=weldPlate_1;
        MoveL Target_1040,v20,z1,Tooldata_1\WObj:=weldPlate_1;
        MoveL Target_1050,v20,z1,Tooldata_1\WObj:=weldPlate_1;
        MoveL Target_1060,v20,z1,Tooldata_1\WObj:=weldPlate_1;
        MoveL Target_1070,v20,z1,Tooldata_1\WObj:=weldPlate_1;
        MoveL Target_1080,v20,z1,Tooldata_1\WObj:=weldPlate_1;
        MoveL Target_1090,v20,z1,Tooldata_1\WObj:=weldPlate_1;
        MoveL Target_1100,v20,z1,Tooldata_1\WObj:=weldPlate_1;
        MoveL Target_1110,v20,z1,Tooldata_1\WObj:=weldPlate_1;
        MoveL Target_1120,v20,z1,Tooldata_1\WObj:=weldPlate_1;
        MoveL Target_1130,v20,z1,Tooldata_1\WObj:=weldPlate_1;
        MoveL Target_1140,v20,z1,Tooldata_1\WObj:=weldPlate_1;
        MoveL Target_1150,v20,z1,Tooldata_1\WObj:=weldPlate_1;
        MoveL Target_1160,v20,z1,Tooldata_1\WObj:=weldPlate_1;
        MoveL Target_1170,v20,z1,Tooldata_1\WObj:=weldPlate_1;
        MoveL Target_1180,v20,z1,Tooldata_1\WObj:=weldPlate_1;
        MoveL Target_1190,v20,z1,Tooldata_1\WObj:=weldPlate_1;
        MoveL Target_1200,v20,z1,Tooldata_1\WObj:=weldPlate_1;
        MoveL Target_1210,v20,z1,Tooldata_1\WObj:=weldPlate_1;
        MoveL Target_1220,v20,z1,Tooldata_1\WObj:=weldPlate_1;
        MoveL Target_1230,v20,z1,Tooldata_1\WObj:=weldPlate_1;
        MoveL Target_1240,v20,z1,Tooldata_1\WObj:=weldPlate_1;
        MoveL Target_1250,v20,z1,Tooldata_1\WObj:=weldPlate_1;
        MoveL Target_40,v20,z1,Tooldata_1\WObj:=weldPlate_1;
        MoveL Target_50,v20,z1,Tooldata_1\WObj:=weldPlate_1;
        MoveL Target_60,v20,z1,Tooldata_1\WObj:=weldPlate_1;
        MoveL Target_70,v20,z1,Tooldata_1\WObj:=weldPlate_1;
        MoveL Target_70_2,v20,z1,Tooldata_1\WObj:=weldPlate_1;
        MoveL Target_70_2_2,v20,z1,Tooldata_1\WObj:=weldPlate_1;
        MoveL Target_70_3,v20,z1,Tooldata_1\WObj:=weldPlate_1;
        MoveL Target_80,v20,z1,Tooldata_1\WObj:=weldPlate_1;
        MoveL Target_80_3,v20,z1,Tooldata_1\WObj:=weldPlate_1;
        MoveL Target_80_4,v20,z1,Tooldata_1\WObj:=weldPlate_1;
        MoveL Target_90,v20,z1,Tooldata_1\WObj:=weldPlate_1;
        MoveL Target_100,v20,z1,Tooldata_1\WObj:=weldPlate_1;
        MoveL Target_100_3,v20,z1,Tooldata_1\WObj:=weldPlate_1;
        MoveL Target_110,v20,z1,Tooldata_1\WObj:=weldPlate_1;
        MoveL Target_120,v20,z1,Tooldata_1\WObj:=weldPlate_1;
        MoveL Target_120_3,v20,z1,Tooldata_1\WObj:=weldPlate_1;
        MoveL Target_130,v20,z1,Tooldata_1\WObj:=weldPlate_1;
        MoveL Target_140,v20,z1,Tooldata_1\WObj:=weldPlate_1;
        MoveL zEnd_Point,v20,z1,Tooldata_1\WObj:=weldPlate_1;
    ENDPROC
ENDMODULE
